SUBAPPLICATION Uebung_083 (* Beispiel für E_CTUD_UDINT *)
  (* Standard: 61499-2; Description: Copyright (c) 2023 Meisterschulen am Ostbahnhof This program and the accompanying materials are made available under the terms of the Eclipse Public License 2.0 which is available at https://www.eclipse.org/legal/epl-2.0/ SPDX-License-Identifier: EPL-2.0 *)
  (* Version 1.0, 2023-10-23, Franz Höpfinger, Meisterschulen am Ostbahnhof, initial API and implementation and/or initial documentation *)
  PACKAGE Uebungen;
  IMPORT Uebungen::const::UT::DefaultPool::OutputNumber_N1;
  IMPORT logiBUS::io::DI::logiBUS_DI::Input_I1;
  IMPORT logiBUS::io::DI::logiBUS_DI::Input_I2;
  IMPORT logiBUS::io::DI::logiBUS_DI::Input_I3;
  IMPORT logiBUS::io::DI::logiBUS_DI::Input_I4;
  IMPORT logiBUS::io::DI::logiBUS_DI_Events::BUTTON_SINGLE_CLICK;
  IMPORT logiBUS::io::DQ::logiBUS_DO::Output_Q1;
  IMPORT logiBUS::io::DQ::logiBUS_DO::Output_Q2;
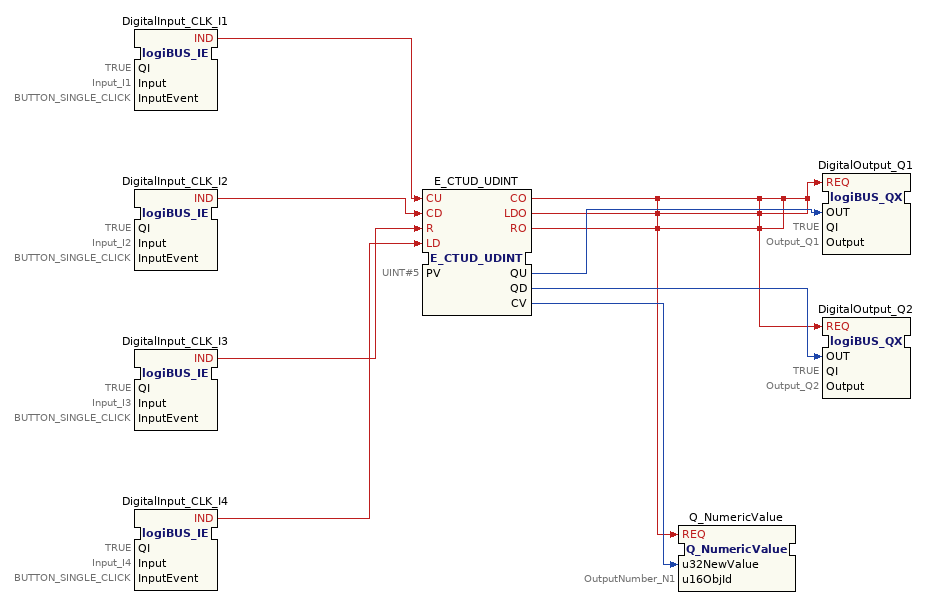
  FBS
    DigitalOutput_Q1 : logiBUS::io::DQ::logiBUS_QX(QI := TRUE, Output := Output_Q1);
    DigitalInput_CLK_I1 : logiBUS::io::DI::logiBUS_IE(QI := TRUE, Input := Input_I1, InputEvent := BUTTON_SINGLE_CLICK);
    E_CTUD_UDINT : iec61499::events::E_CTUD_UDINT(PV := UINT#5);
    DigitalInput_CLK_I2 : logiBUS::io::DI::logiBUS_IE(QI := TRUE, Input := Input_I2, InputEvent := BUTTON_SINGLE_CLICK);
    DigitalInput_CLK_I3 : logiBUS::io::DI::logiBUS_IE(QI := TRUE, Input := Input_I3, InputEvent := BUTTON_SINGLE_CLICK);
    DigitalInput_CLK_I4 : logiBUS::io::DI::logiBUS_IE(QI := TRUE, Input := Input_I4, InputEvent := BUTTON_SINGLE_CLICK);
    DigitalOutput_Q2 : logiBUS::io::DQ::logiBUS_QX(QI := TRUE, Output := Output_Q2);
    Q_NumericValue : isobus::UT::Q::Q_NumericValue(u16ObjId := OutputNumber_N1);
  END_FBS
  EVENT_CONNECTIONS
    DigitalInput_CLK_I1.IND TO E_CTUD_UDINT.CU;
    E_CTUD_UDINT.CO TO DigitalOutput_Q1.REQ;
    E_CTUD_UDINT.LDO TO DigitalOutput_Q1.REQ;
    DigitalInput_CLK_I2.IND TO E_CTUD_UDINT.CD;
    E_CTUD_UDINT.RO TO DigitalOutput_Q1.REQ;
    DigitalInput_CLK_I3.IND TO E_CTUD_UDINT.R;
    DigitalInput_CLK_I4.IND TO E_CTUD_UDINT.LD;
    E_CTUD_UDINT.LDO TO DigitalOutput_Q2.REQ;
    E_CTUD_UDINT.CO TO DigitalOutput_Q2.REQ;
    E_CTUD_UDINT.RO TO DigitalOutput_Q2.REQ;
    E_CTUD_UDINT.CO TO Q_NumericValue.REQ;
    E_CTUD_UDINT.RO TO Q_NumericValue.REQ;
    E_CTUD_UDINT.LDO TO Q_NumericValue.REQ;
  END_CONNECTIONS
  DATA_CONNECTIONS
    E_CTUD_UDINT.QU TO DigitalOutput_Q1.OUT;
    E_CTUD_UDINT.QD TO DigitalOutput_Q2.OUT;
    E_CTUD_UDINT.CV TO Q_NumericValue.u32NewValue;
  END_CONNECTIONS
END_SUBAPPLICATION
